{attribute 'qualified_only'}
VAR_GLOBAL
	bStart : BOOL;
	nCount : INT ;
END_VAR

(* stored: Version 1.1.0.1, ProductVersion 3.1.4024.16
   GVL GVL: Id {5b5fbd45-af47-4d96-8dac-e9aa78c3cedb} *)
